Staubli VAL3: RefreshList.pgx

program RefreshList()
  local num l_ni
begin
  //
  switch nPage
    case 0
      if bListRefresh
        resize(sList,1,size(sPrd))
        for l_ni=0 to size(sList)-1
          sList[l_ni]=sPrd[l_ni]
        endFor
      endIf
    break
    case 1
      resize(sList,1,size(sPathList))
      for l_ni=0 to size(sList)-1
        sList[l_ni]=sPathList[l_ni]
      endFor
    break
    //
    case 2
      resize(sList,1,size(sFileList))
        for l_ni=0 to size(sList)-1
          sList[l_ni]=sFileList[l_ni]
        endFor
    break
  endSwitch
end
